TYPE E_MoveState :
(
	ABORT,
	INIT,
	ENABLE,
	FORWARD,
	BACKWARDS,
	READY,
	MOVING,
	NEWTARGETPOSITION,
	NEWTARGETPOSITION2,
	ERROR,
	RESET,
	HALT,
	HOME
) UDINT;
END_TYPE

(* stored: Version 1.1.0.1, ProductVersion 3.1.4024.3
   DUT E_MoveState: Id {3c0d4f9f-7faf-4139-8fac-b742d44134cd} *)
